FUNCTION_BLOCK FB_PID
VAR
	bSync			: BOOL;					(* Synchronize controller							*)
	bSyncSR			: RS;					(* Set reset synchronize controller					*)
	bSyncMaxTime	: TON;					(* Timer for max synchronisation time				*)

	bHoldLocal		: BOOL;					(* Internal hold bit								*)

	eMode			: E_CTRL_MODE;			(* Controller mode									*)
	eState			: E_CTRL_STATE;			(* Controller mode: passive, activ, check, error 	*)

	stParams	: ST_CTRL_PID_EXT_PARAMS;	(* controller External PID parameters				*)

	PID_EXT		: FB_CTRL_PID_EXT;			(* PID controller									*)
	PID_ROC		: FB_PID_ROC;				(* PID rate of change								*)

	bMaxLimitReached	: BOOL := FALSE;	(* Minimum limiting active ? [TRUE/FALSE] -> ARW 	*)
	bMinLimitReached	: BOOL := FALSE;	(* Maximum limiting active ? [TRUE/FALSE] -> ARW 	*)
	bARWActive			: BOOL := FALSE;	(* ARW actice ? [TRUE/FALSE] -> freeze I-part		*)

	ManualFTRIG			: F_TRIG;			(* Trigger for manual mode							*)

	(* auxiliary outputs *)
	fCtrlDerivation		: REAL; 			(* Controller command derivation dy/dt				 *)
	ROCIN				: REAL;				(* Value rate of change input						*)


	(* error outputs *)
	bError				: BOOL;					(* error flag 					*)
	eErrorId			: E_CTRL_ERRORCODES;	(* error code 					*)
	PID_fOut			: REAL;					(* error pid value output		*)
	fOut_Old			: REAL;					(* error value old output value	*)
END_VAR

VAR_INPUT
	bEnable				: BOOL;	(* controller enabled 				*)
	bReset				: BOOL;	(* reset controller 				*)
	bMAn_On				: BOOL;	(* controller in manual				*)
	bHold				: BOOL;	(* hold values						*)
	fOutput_Min			: REAL;	(* minimum value output				*)
	fOutput_Max			: REAL;	(* maximum value output				*)
	fOutput_ROC_Up		: REAL; (* Rate of change value output up	*)
	fOutput_ROC_Dn		: REAL; (* Rate of change value output down	*)
	fKp					: REAL;	(* Proportional value				*)
	tTn					: TIME;	(* Timer Tn time					*)
	tTv					: TIME;	(* Timer Tv time					*)
	tTd					: TIME;	(* Timer Td time					*)
	fDeadBandInput		: REAL;	(* input value deadband				*)
	fI_InnerWindow		: REAL;	(* value inner window				*)
	fSetpoint			: REAL;	(* setpoint value					*)
	fActual				: REAL;	(* actual value						*)
	fMAnValue			: REAL;	(* manual value						*)

	tTaskCycleTime		: TIME;	(* task cycle time					*)
	tCtrlCycleTime		: TIME;	(* control cycle time				*)

END_VAR

VAR_OUTPUT
	fOut				: REAL;	(* output value						*)
END_VAR

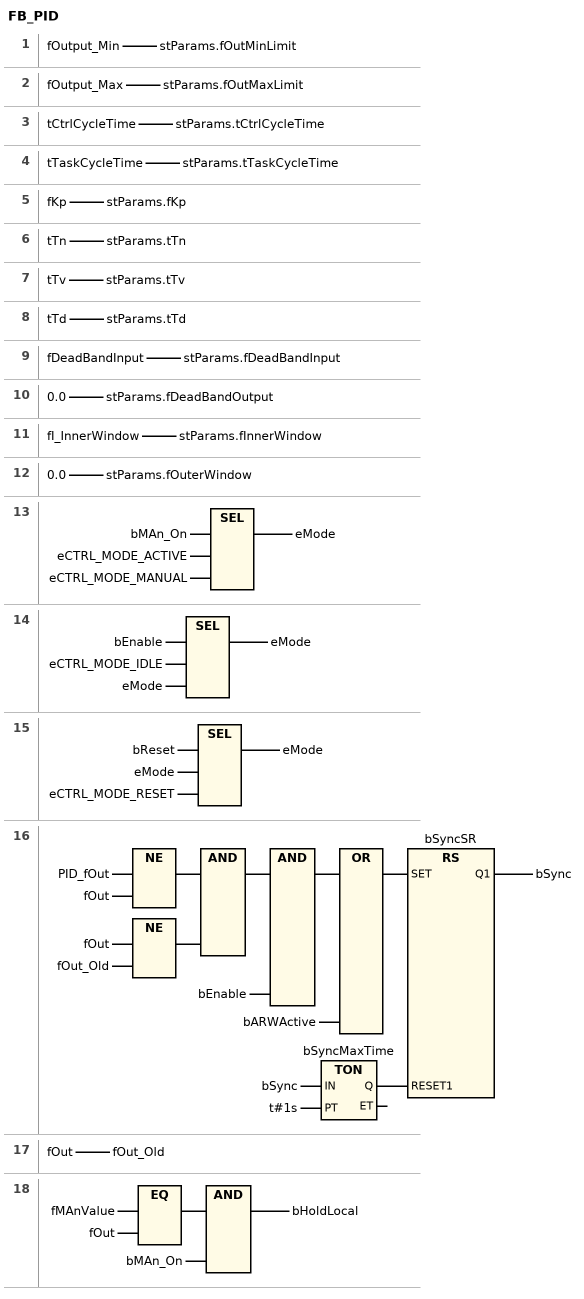
// NETWORK 1
stParams.fOutMinLimit := fOutput_Min;

// NETWORK 2
stParams.fOutMaxLimit := fOutput_Max;

// NETWORK 3
stParams.tCtrlCycleTime := tCtrlCycleTime;

// NETWORK 4
stParams.tTaskCycleTime := tTaskCycleTime;

// NETWORK 5
stParams.fKp := fKp;

// NETWORK 6
stParams.tTn := tTn;

// NETWORK 7
stParams.tTv := tTv;

// NETWORK 8
stParams.tTd := tTd;

// NETWORK 9
stParams.fDeadBandInput := fDeadBandInput;

// NETWORK 10
stParams.fDeadBandOutput := 0.0;

// NETWORK 11
stParams.fInnerWindow := fI_InnerWindow;

// NETWORK 12
stParams.fOuterWindow := 0.0;

// NETWORK 13
eMode := SEL(bMAn_On, eCTRL_MODE_ACTIVE, eCTRL_MODE_MANUAL);

// NETWORK 14
eMode := SEL(bEnable, eCTRL_MODE_IDLE, eMode);

// NETWORK 15
eMode := SEL(bReset, eMode, eCTRL_MODE_RESET);

// NETWORK 16
bSyncMaxTime(IN := bSync, PT := t#1s); // TON
bSyncSR(SET := (PID_fOut <> fOut AND fOut <> fOut_Old) AND bEnable OR bARWActive, RESET1 := bSyncMaxTime.Q); // RS
bSync := bSyncSR.Q1;

// NETWORK 17
fOut_Old := fOut;

// NETWORK 18
bHoldLocal := fMAnValue = fOut AND bMAn_On;

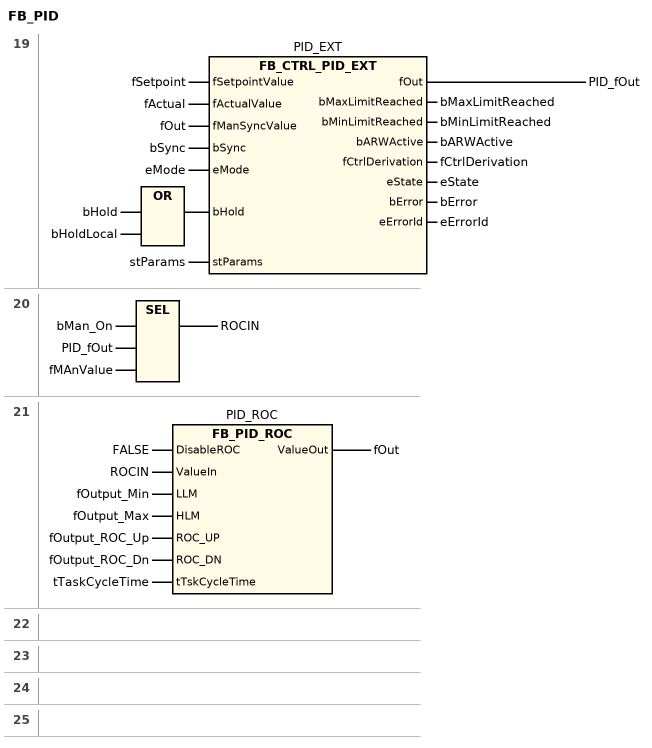
// NETWORK 19
PID_EXT(
    fSetpointValue := fSetpoint,
    fActualValue := fActual,
    fManSyncValue := fOut,
    bSync := bSync,
    eMode := eMode,
    bHold := bHold OR bHoldLocal,
    stParams := stParams,
    bMaxLimitReached => bMaxLimitReached,
    bMinLimitReached => bMinLimitReached,
    bARWActive => bARWActive,
    fCtrlDerivation => fCtrlDerivation,
    eState => eState,
    bError => bError,
    eErrorId => eErrorId); // FB_CTRL_PID_EXT
PID_fOut := PID_EXT.fOut;

// NETWORK 20
ROCIN := SEL(bMan_On, PID_fOut, fMAnValue);

// NETWORK 21
PID_ROC(
    DisableROC := FALSE,
    ValueIn := ROCIN,
    LLM := fOutput_Min,
    HLM := fOutput_Max,
    ROC_UP := fOutput_ROC_Up,
    ROC_DN := fOutput_ROC_Dn,
    tTskCycleTime := tTaskCycleTime); // FB_PID_ROC
fOut := PID_ROC.ValueOut;

// NETWORK 22

// NETWORK 23

// NETWORK 24

// NETWORK 25

END_FUNCTION_BLOCK

(* stored: Version 1.1.0.1, ProductVersion 3.1.4020.12
   POU FB_PID: Id {93a4746c-b478-446e-85b0-7c060575e2f6}, SpecialFunc None *)
